FUNCTION F_ToAnyString : T_AnyString
VAR_INPUT
    anyArg	: ANY_STRING;
END_VAR

F_ToAnyString := anyArg;

END_FUNCTION

(* stored: Version 1.1.0.1
   POU F_ToAnyString: Id {32964a37-44f5-4640-96f6-05e873239ad6}, SpecialFunc None *)
